{attribute 'qualified_only'}
{attribute 'strict'}
{attribute 'to_string'}
TYPE E_MachineState :
(
	PowerUp := 0,
    Fault,
    Stopping,
    Stopped,
    Initialising,
    ReadyToStart,
    AutoCycle,
    Manual
);
END_TYPE

(* stored: Version 1.1.0.1, ProductVersion 3.1.4026.18
   DUT E_MachineState: Id {473e1156-2b87-40d4-a57b-c37602246c60} *)
